{attribute 'qualified_only'}
VAR_GLOBAL
	Logger	: ZigaLibs_Logging.FB_Logger;
	ILogger	: ZigaLibs_Core.I_LoggerEx := Logger;
END_VAR

(* stored: Version 1.1.0.1, ProductVersion 3.1.4024.14
   GVL GVL: Id {008c5c7c-3d8c-060a-0cee-56c6b0a37b30} *)
